TYPE DUT_Recipe_Step :
STRUCT
    Step_Name               : STRING(40);
    Target_Power_kW         : REAL;
    Duration                : TIME;
    Enabled                 : BOOL := TRUE;
END_STRUCT
END_TYPE

(* stored: Version 1.1.0.1, ProductVersion 3.1.4024.16
   DUT DUT_Recipe_Step: Id {3b9a94e1-f58d-444d-8a89-06b5f403bd51} *)
